FUNCTION SPLIT_LWORD_INTO_WORDS (* this Function extracts the 4 WORDS from a lword *)
  (* Standard: 61499-1; Description: Copyright (c) 2026 HR Agrartechnik GmbH This program and the accompanying materials are made available under the terms of the Eclipse Public License 2.0 which is available at https://www.eclipse.org/legal/epl-2.0/ SPDX-License-Identifier: EPL-2.0 *)
  (* Version 1.0, 2026-05-16, Franz Höpfinger, HR Agrartechnik, initial Implementation *)
  PACKAGE eclipse4diac::utils::splitting;
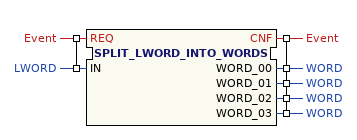
  EVENT_INPUT
    REQ WITH IN;
  END_EVENT
  EVENT_OUTPUT
    CNF WITH WORD_00, WORD_01, WORD_02, WORD_03;
  END_EVENT
  VAR_INPUT
    IN : LWORD;
  END_VAR
  VAR_OUTPUT
    WORD_00 : WORD;
    WORD_01 : WORD;
    WORD_02 : WORD;
    WORD_03 : WORD;
  END_VAR
  BODY IN ST:
PACKAGE eclipse4diac::utils::splitting;

(* this Function extracts the 4 WORDS from a lword *)
FUNCTION SPLIT_LWORD_INTO_WORDS

VAR_INPUT
	IN : LWORD;
END_VAR

VAR_OUTPUT
	WORD_00 : WORD;
	WORD_01 : WORD;
	WORD_02 : WORD;
	WORD_03 : WORD;
END_VAR

WORD_00 := IN.%W0;
WORD_01 := IN.%W1;
WORD_02 := IN.%W2;
WORD_03 := IN.%W3;

END_FUNCTION
  END_BODY
END_FUNCTION
